# EPICS IOC start-up script: examples/test/PSI/MCAG001/new.iocsh
require ecmccfg v8_RC1, "ECMC_VER=v8_RC1,EC_RATE=500"
#require ECMC_EXTRA kivel

epicsEnvSet("DEV", "X00AA-FOO-BAR")

${SCRIPTEXEC} ${ECMC_CONFIG_ROOT}addSlave.cmd,       "HW_DESC=EK1100"

${SCRIPTEXEC} ${ECMC_CONFIG_ROOT}addSlave.cmd,       "HW_DESC=EL1018"

${SCRIPTEXEC} ${ECMC_CONFIG_ROOT}addSlave.cmd,       "HW_DESC=EL2808"
# Set all outputs to feed switches
ecmcConfigOrDie "Cfg.WriteEcEntryIDString(${ECMC_EC_SLAVE_NUM},binaryOutput01,1)"
ecmcConfigOrDie "Cfg.WriteEcEntryIDString(${ECMC_EC_SLAVE_NUM},binaryOutput02,1)"
ecmcConfigOrDie "Cfg.WriteEcEntryIDString(${ECMC_EC_SLAVE_NUM},binaryOutput03,1)"
ecmcConfigOrDie "Cfg.WriteEcEntryIDString(${ECMC_EC_SLAVE_NUM},binaryOutput04,1)"
ecmcConfigOrDie "Cfg.WriteEcEntryIDString(${ECMC_EC_SLAVE_NUM},binaryOutput05,1)"
ecmcConfigOrDie "Cfg.WriteEcEntryIDString(${ECMC_EC_SLAVE_NUM},binaryOutput06,1)"
ecmcConfigOrDie "Cfg.WriteEcEntryIDString(${ECMC_EC_SLAVE_NUM},binaryOutput07,1)"
ecmcConfigOrDie "Cfg.WriteEcEntryIDString(${ECMC_EC_SLAVE_NUM},binaryOutput08,1)"

#- top axis
${SCRIPTEXEC} ${ECMC_CONFIG_ROOT}addSlave.cmd,       "HW_DESC=EL5101"
# Reverse encoder direction:
ecmcConfigOrDie "Cfg.EcAddSdo(${ECMC_EC_SLAVE_NUM},0x8010,0x0e,1,1)"
${SCRIPTEXEC} ${ecmccfg_DIR}configureSlave.cmd, "HW_DESC=EL7037, CONFIG=-Motor-Nanotec-ST4118L1804-B"
# Reverse motor direction:
ecmcConfigOrDie "Cfg.EcAddSdo(${ECMC_EC_SLAVE_NUM},0x8012,0x9,1,1)"

#- #############################################################################
#- apply configuration
${SCRIPTEXEC} ${ECMC_CONFIG_ROOT}applyConfig.cmd
#- #############################################################################
#- go active
${SCRIPTEXEC} ${ecmccfg_DIR}setAppMode.cmd
